Xinje XCPPro project, PLC1: XC3-14 (software 3.3r 2017-11-30)

PROGRAM Ladder

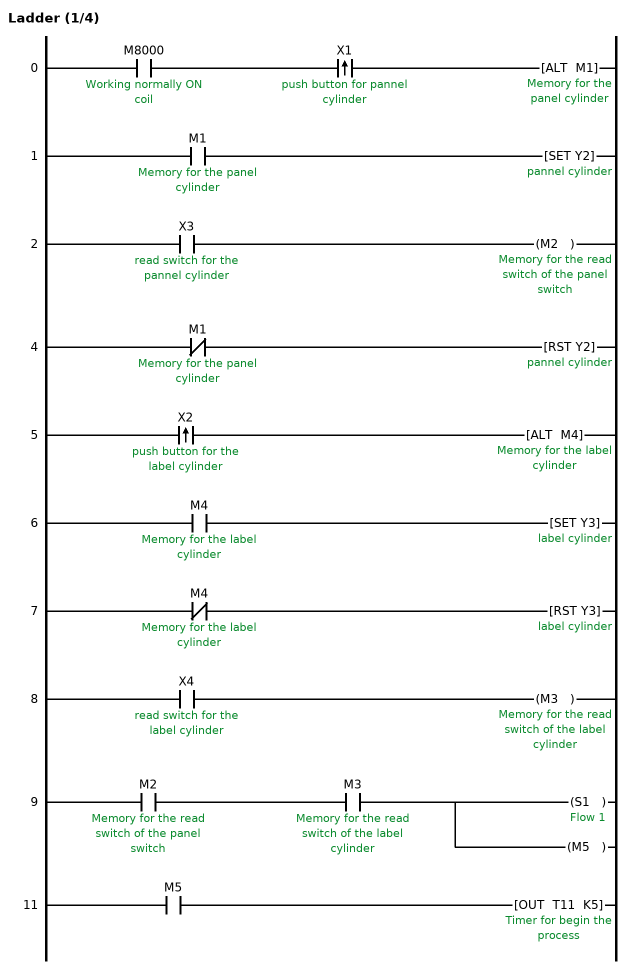
LD     M8000	; Working normally ON coil
ANDP   X1	; push button for pannel cylinder
ALT    M1	; Memory for the panel cylinder
LD     M1	; Memory for the panel cylinder
SET    Y2	; pannel cylinder
LD     X3	; read switch for the pannel cylinder
OUT    M2	; Memory for the read switch of the panel switch
LDI    M1	; Memory for the panel cylinder
RST    Y2	; pannel cylinder
LDP    X2	; push button for the label cylinder
ALT    M4	; Memory for the label cylinder
LD     M4	; Memory for the label cylinder
SET    Y3	; label cylinder
LDI    M4	; Memory for the label cylinder
RST    Y3	; label cylinder
LD     X4	; read switch for the label cylinder
OUT    M3	; Memory for the read switch of the label cylinder
LD     M2	; Memory for the read switch of the panel switch
AND    M3	; Memory for the read switch of the label cylinder
OUT    S1	; Flow 1
OUT    M5
LD     M5
OUT    T11 K5	; Timer for begin the process

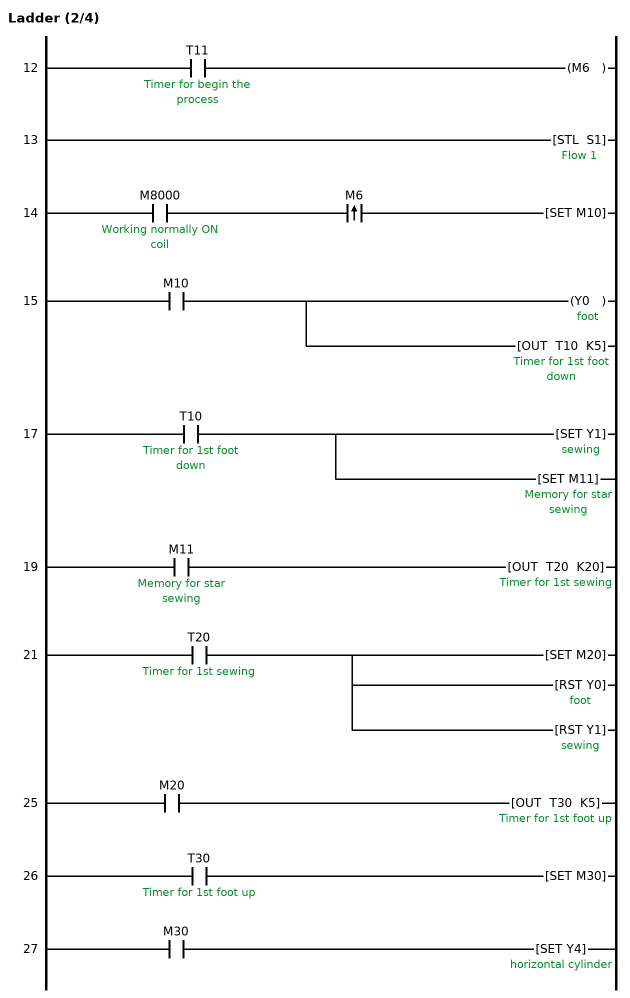
LD     T11	; Timer for begin the process
OUT    M6
STL    S1	; Flow 1
LD     M8000	; Working normally ON coil
ANDP   M6
SET    M10
LD     M10
OUT    Y0	; foot
OUT    T10 K5	; Timer for 1st foot down
LD     T10	; Timer for 1st foot down
SET    Y1	; sewing
SET    M11	; Memory for star sewing
LD     M11	; Memory for star sewing
OUT    T20 K20	; Timer for 1st sewing
LD     T20	; Timer for 1st sewing
SET    M20
RST    Y0	; foot
RST    Y1	; sewing
LD     M20
OUT    T30 K5	; Timer for 1st foot up
LD     T30	; Timer for 1st foot up
SET    M30
LD     M30
SET    Y4	; horizontal cylinder

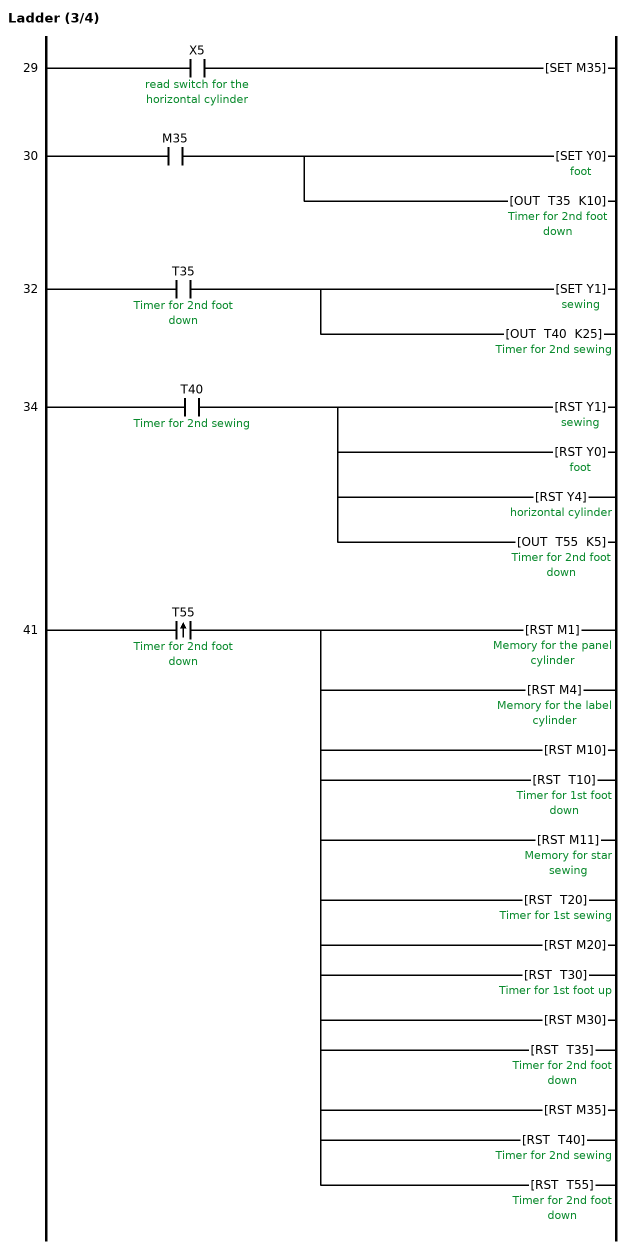
LD     X5	; read switch for the horizontal cylinder
SET    M35
LD     M35
SET    Y0	; foot
OUT    T35 K10	; Timer for 2nd foot down
LD     T35	; Timer for 2nd foot down
SET    Y1	; sewing
OUT    T40 K25	; Timer for 2nd sewing
LD     T40	; Timer for 2nd sewing
RST    Y1	; sewing
RST    Y0	; foot
RST    Y4	; horizontal cylinder
OUT    T55 K5	; Timer for 2nd foot down
LDP    T55	; Timer for 2nd foot down
RST    M1	; Memory for the panel cylinder
RST    M4	; Memory for the label cylinder
RST    M10
RST    T10	; Timer for 1st foot down
RST    M11	; Memory for star sewing
RST    T20	; Timer for 1st sewing
RST    M20
RST    T30	; Timer for 1st foot up
RST    M30
RST    T35	; Timer for 2nd foot down
RST    M35
RST    T40	; Timer for 2nd sewing
RST    T55	; Timer for 2nd foot down

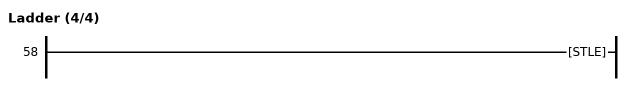
STLE